FUNCTION_BLOCK FB_LogowanieBledow
VAR_INPUT
END_VAR
VAR_OUTPUT
END_VAR
VAR
	tablica 								: ARRAY [1..GVL_LogowanieBledow_Stale.MAX_ILOSC_ELEMENTOW] OF ITF_LogowanieBledow_ElementWykonawczy;
	iIloscDodanychElementow					: INT;
	iID 									: INT;	//ilosść dodanych zdarzeń globalnie
	iJezykID								: INT := 1045;	//id języka - domyślnie polski
	bwypelnij								: BOOL;		//Wypełnienie tablic - wykonać na początku i po zmianie języka
	bDaneWypelnione							: BOOL := FALSE;	//jak true mozna odczytywac stany podzespolow
	iI										: INT;
	iJ										: INT;
	
	arrTablicaDefinicjiZdarzen				: ARRAY [1..GVL_LogowanieBledow_Stale.MAX_ILOSC_ZDARZEN] OF DUT_LogowanieBledow_Zdarzenie;
	arrTablicaDefinicjiZdarzenOpis			: ARRAY [1..GVL_LogowanieBledow_Stale.MAX_ILOSC_ZDARZEN] OF DUT_LogowanieBledow_ZdarzenieOpis;
	arrTablicaDefinicjiZdarzenStan			: ARRAY [1..GVL_LogowanieBledow_Stale.MAX_ILOSC_ZDARZEN] OF DUT_LogowanieBledow_ZdarzenieStan;

END_VAR

//Wypełnienie tablicy zdarzen dla wszystkich elementow
	IF(bwypelnij) THEN
		bDaneWypelnione						:= FALSE;
		FOR iI := 1 TO iIloscDodanychElementow DO 
			tablica [iI].ZwrocTabliceDefinicji (	arrTablicaDefinicjiZdarzen := arrTablicaDefinicjiZdarzen,
													arrTablicaDefinicjiZdarzenOpis := arrTablicaDefinicjiZdarzenOpis,
													arrTablicaDefinicjiZdarzenStan := arrTablicaDefinicjiZdarzenStan,
													iIdZdarzenia := iID, 
													iNrPodzespolu := iI, 
													iNrPodelementu := 1,
													iNrElementu := 1, 
													iJezykId := iJezykID);
		END_FOR
		bwypelnij := FALSE;
		bDaneWypelnione						:= TRUE;
	END_IF

//Aktualizacja tablicy stanów
	IF (bDaneWypelnione) THEN
		FOR iJ := 1 TO iIloscDodanychElementow DO
			tablica [iJ].ZwrocTabliceStanu (arrTablicaDefinicjiZdarzenStan := arrTablicaDefinicjiZdarzenStan);
		END_FOR
	END_IF

METHOD FB_init : BOOL
VAR_INPUT
	bInitRetains : BOOL; // if TRUE, the retain variables are initialized (warm start / cold start)
	bInCopyCode : BOOL;  // if TRUE, the instance afterwards gets moved into the copy code (online change)
	tablica 								: ARRAY [1..GVL_LogowanieBledow_Stale.MAX_ILOSC_ELEMENTOW] OF ITF_LogowanieBledow_ElementWykonawczy;
	iIloscDodanychElementow					: INT;
END_VAR
THIS^.tablica 								:= tablica;
THIS^.iIloscDodanychElementow				:= iIloscDodanychElementow;
END_METHOD

PROPERTY WypelnijTabliceZdarzen : BOOL
SET
bwypelnij									:= WypelnijTabliceZdarzen;
END_SET
END_PROPERTY

END_FUNCTION_BLOCK

(* stored: Version 1.1.0.1, ProductVersion 3.1.4024.11
   POU FB_LogowanieBledow: Id {b71b0a28-4386-4dc4-b55c-25a29e40a801}, SpecialFunc None
   Method FB_init: Id {b7e0c430-8f48-483d-850f-546111d97dba}
   Property WypelnijTabliceZdarzen: Id {4a058b9b-7ed5-4a20-8f86-36e7cd0888e3}
   Set Set: Id {432c778d-56b7-467a-8279-dc1872be0bc5} *)
